// Mitsubishi GX Works2 project: Genova 14-11-2022_f1   PLC: FX1N/FX1NC

PROGRAM MAIN
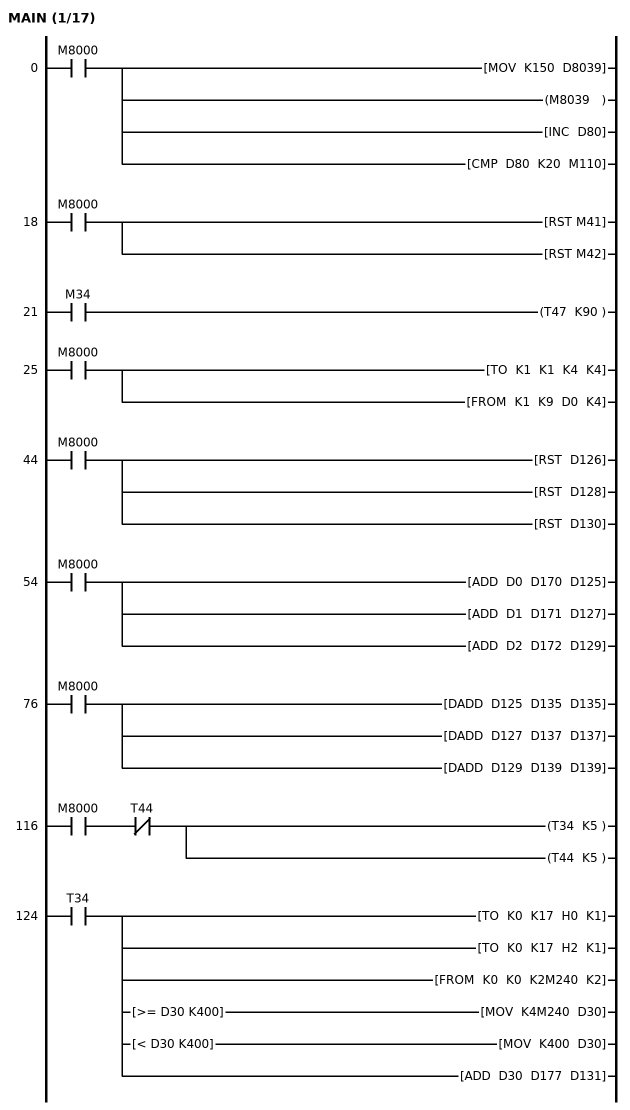
0     LD      M8000
      MOV     K150 D8039
      OUT     M8039
      INC     D80
      CMP     D80 K20 M110
18    LD      M8000
      RST     M41
      RST     M42
21    LD      M34
      OUT     T47 K90
25    LD      M8000
      TO      K1 K1 K4 K4
      FROM    K1 K9 D0 K4
44    LD      M8000
      RST     D126
      RST     D128
      RST     D130
54    LD      M8000
      ADD     D0 D170 D125
      ADD     D1 D171 D127
      ADD     D2 D172 D129
76    LD      M8000
      DADD    D125 D135 D135
      DADD    D127 D137 D137
      DADD    D129 D139 D139
116   LD      M8000
      ANI     T44
      OUT     T34 K5
      OUT     T44 K5
124   LD      T34
      TO      K0 K17 H0 K1
      TO      K0 K17 H2 K1
      FROM    K0 K0 K2M240 K2
      MPS
      AND>=   D30 K400
      MOV     K4M240 D30
      MRD
      AND<    D30 K400
      MOV     K400 D30
      MPP
      ADD     D30 D177 D131
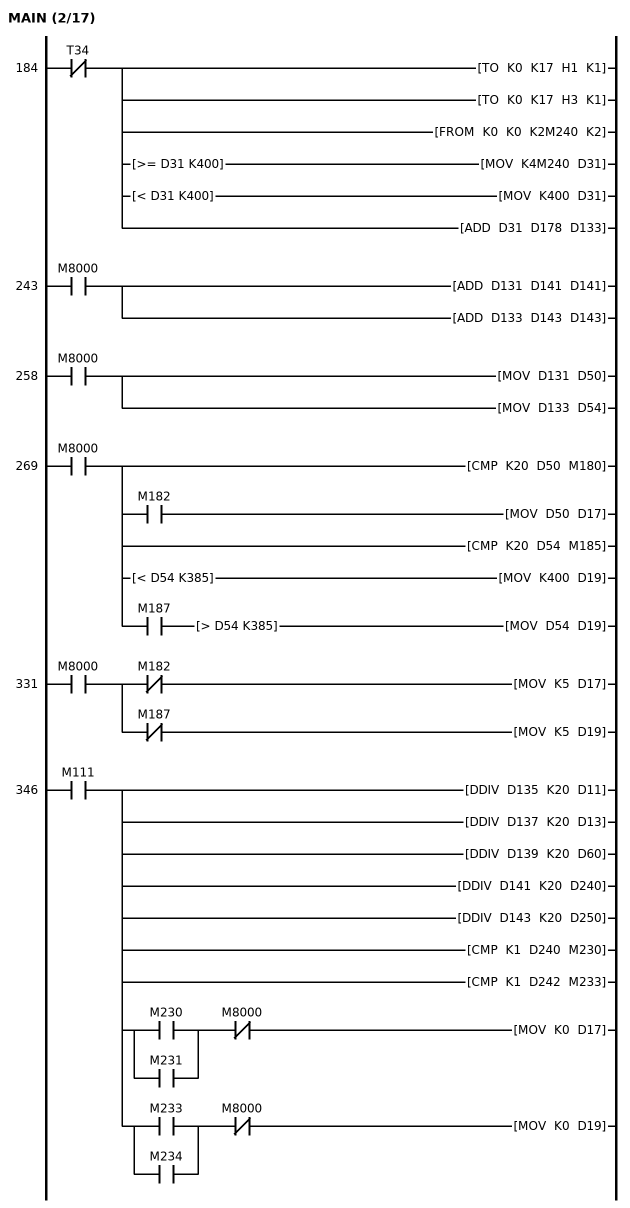
184   LDI     T34
      TO      K0 K17 H1 K1
      TO      K0 K17 H3 K1
      FROM    K0 K0 K2M240 K2
      MPS
      AND>=   D31 K400
      MOV     K4M240 D31
      MRD
      AND<    D31 K400
      MOV     K400 D31
      MPP
      ADD     D31 D178 D133
243   LD      M8000
      ADD     D131 D141 D141
      ADD     D133 D143 D143
258   LD      M8000
      MOV     D131 D50
      MOV     D133 D54
269   LD      M8000
      CMP     K20 D50 M180
      MPS
      AND     M182
      MOV     D50 D17
      MPP
      CMP     K20 D54 M185
      MPS
      AND<    D54 K385
      MOV     K400 D19
      MPP
      AND     M187
      AND>    D54 K385
      MOV     D54 D19
331   LD      M8000
      MPS
      ANI     M182
      MOV     K5 D17
      MPP
      ANI     M187
      MOV     K5 D19
346   LD      M111
      DDIV    D135 K20 D11
      DDIV    D137 K20 D13
      DDIV    D139 K20 D60
      DDIV    D141 K20 D240
      DDIV    D143 K20 D250
      CMP     K1 D240 M230
      CMP     K1 D242 M233
      MPS
      LD      M230
      OR      M231
      ANB
      ANI     M8000
      MOV     K0 D17
      MPP
      LD      M233
      OR      M234
      ANB
      ANI     M8000
      MOV     K0 D19
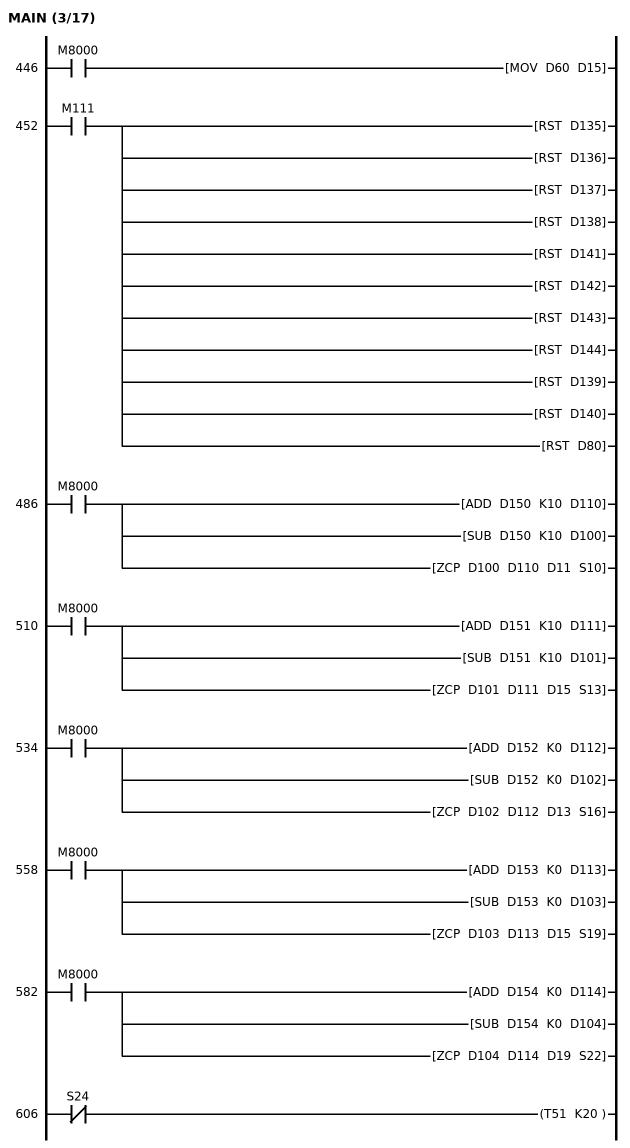
446   LD      M8000
      MOV     D60 D15
452   LD      M111
      RST     D135
      RST     D136
      RST     D137
      RST     D138
      RST     D141
      RST     D142
      RST     D143
      RST     D144
      RST     D139
      RST     D140
      RST     D80
486   LD      M8000
      ADD     D150 K10 D110
      SUB     D150 K10 D100
      ZCP     D100 D110 D11 S10
510   LD      M8000
      ADD     D151 K10 D111
      SUB     D151 K10 D101
      ZCP     D101 D111 D15 S13
534   LD      M8000
      ADD     D152 K0 D112
      SUB     D152 K0 D102
      ZCP     D102 D112 D13 S16
558   LD      M8000
      ADD     D153 K0 D113
      SUB     D153 K0 D103
      ZCP     D103 D113 D15 S19
582   LD      M8000
      ADD     D154 K0 D114
      SUB     D154 K0 D104
      ZCP     D104 D114 D19 S22
606   LDI     S24
      OUT     T51 K20
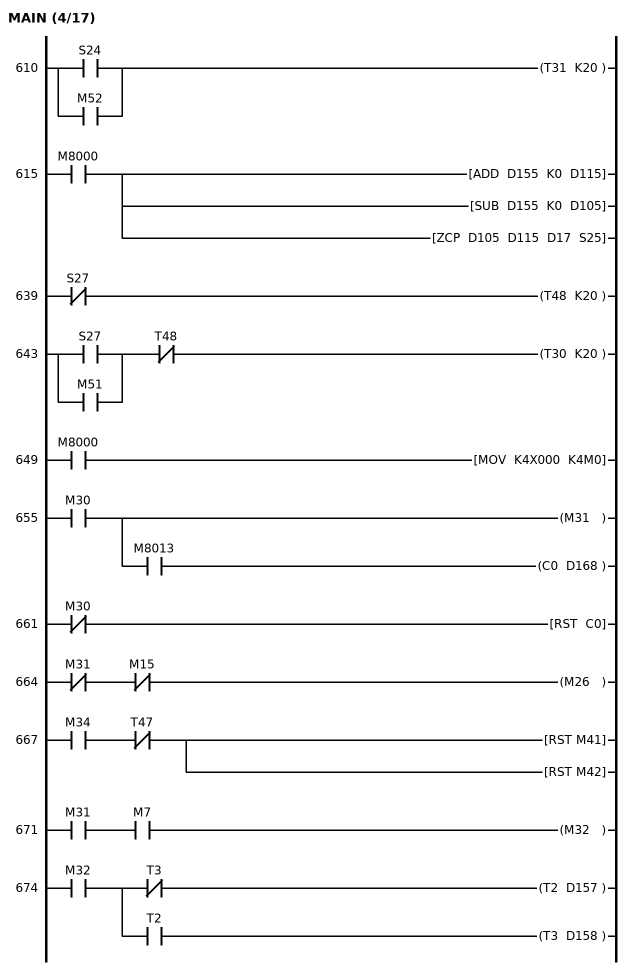
610   LD      S24
      OR      M52
      OUT     T31 K20
615   LD      M8000
      ADD     D155 K0 D115
      SUB     D155 K0 D105
      ZCP     D105 D115 D17 S25
639   LDI     S27
      OUT     T48 K20
643   LD      S27
      OR      M51
      ANI     T48
      OUT     T30 K20
649   LD      M8000
      MOV     K4X000 K4M0
655   LD      M30
      OUT     M31
      AND     M8013
      OUT     C0 D168
661   LDI     M30
      RST     C0
664   LDI     M31
      ANI     M15
      OUT     M26
667   LD      M34
      ANI     T47
      RST     M41
      RST     M42
671   LD      M31
      AND     M7
      OUT     M32
674   LD      M32
      MPS
      ANI     T3
      OUT     T2 D157
      MPP
      AND     T2
      OUT     T3 D158
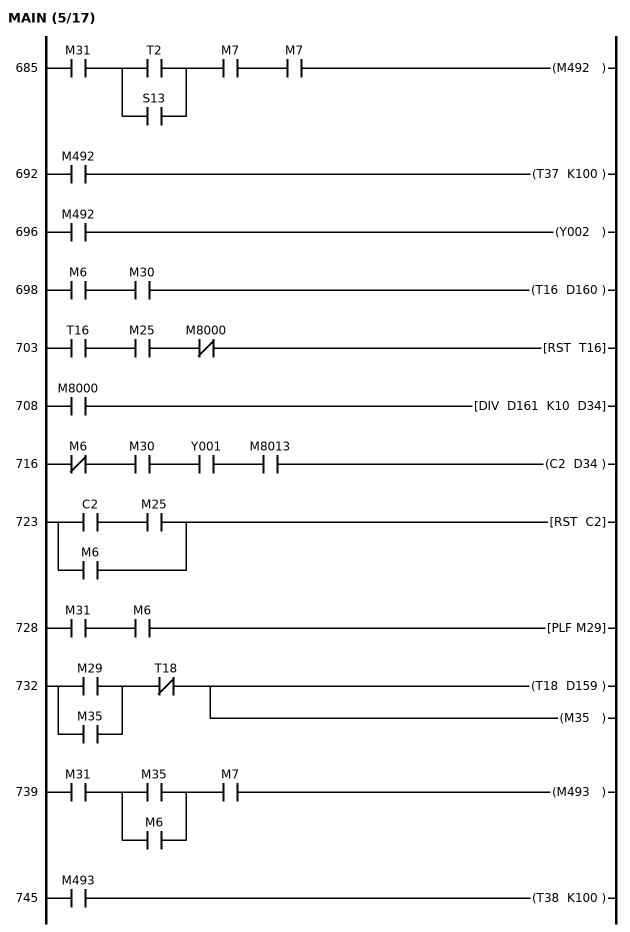
685   LD      M31
      LD      T2
      OR      S13
      ANB
      AND     M7
      AND     M7
      OUT     M492
692   LD      M492
      OUT     T37 K100
696   LD      M492
      OUT     Y002
698   LD      M6
      AND     M30
      OUT     T16 D160
703   LD      T16
      AND     M25
      ANI     M8000
      RST     T16
708   LD      M8000
      DIV     D161 K10 D34
716   LDI     M6
      AND     M30
      AND     Y001
      AND     M8013
      OUT     C2 D34
723   LD      C2
      AND     M25
      OR      M6
      RST     C2
728   LD      M31
      AND     M6
      PLF     M29
732   LD      M29
      OR      M35
      ANI     T18
      OUT     T18 D159
      OUT     M35
739   LD      M31
      LD      M35
      OR      M6
      ANB
      AND     M7
      OUT     M493
745   LD      M493
      OUT     T38 K100
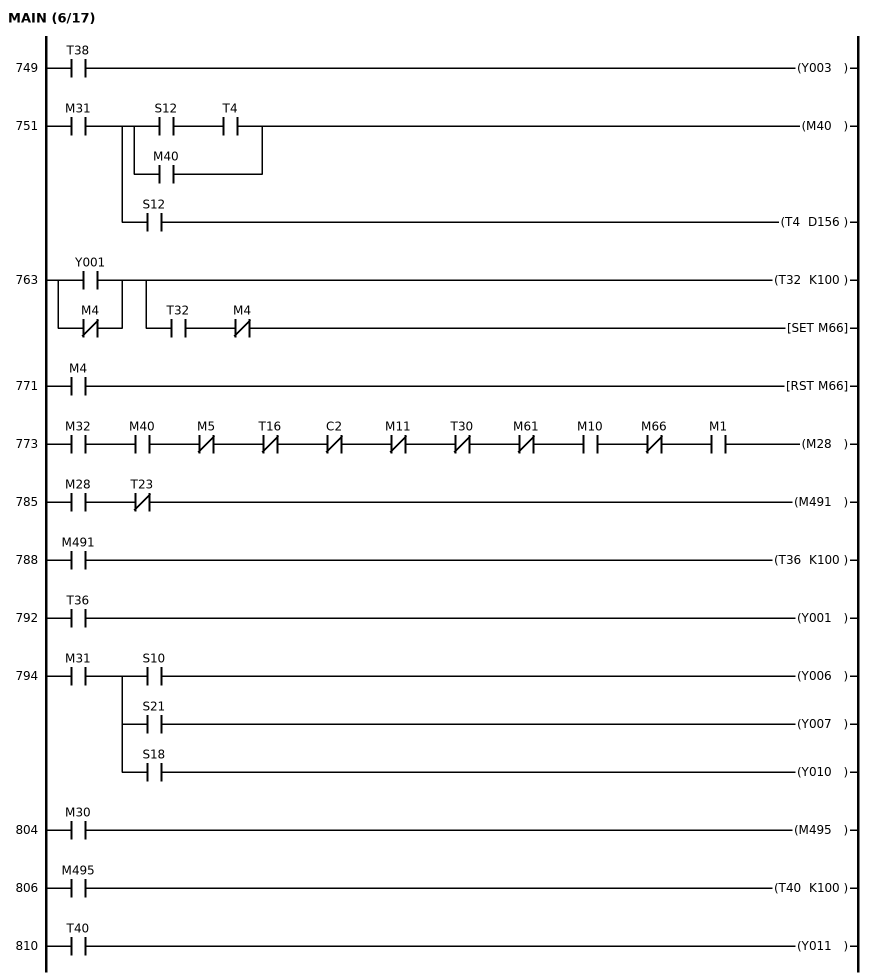
749   LD      T38
      OUT     Y003
751   LD      M31
      MPS
      LD      S12
      AND     T4
      OR      M40
      ANB
      OUT     M40
      MPP
      AND     S12
      OUT     T4 D156
763   LD      Y001
      ORI     M4
      OUT     T32 K100
      AND     T32
      ANI     M4
      SET     M66
771   LD      M4
      RST     M66
773   LD      M32
      AND     M40
      ANI     M5
      ANI     T16
      ANI     C2
      ANI     M11
      ANI     T30
      ANI     M61
      AND     M10
      ANI     M66
      AND     M1
      OUT     M28
785   LD      M28
      ANI     T23
      OUT     M491
788   LD      M491
      OUT     T36 K100
792   LD      T36
      OUT     Y001
794   LD      M31
      MPS
      AND     S10
      OUT     Y006
      MRD
      AND     S21
      OUT     Y007
      MPP
      AND     S18
      OUT     Y010
804   LD      M30
      OUT     M495
806   LD      M495
      OUT     T40 K100
810   LD      T40
      OUT     Y011
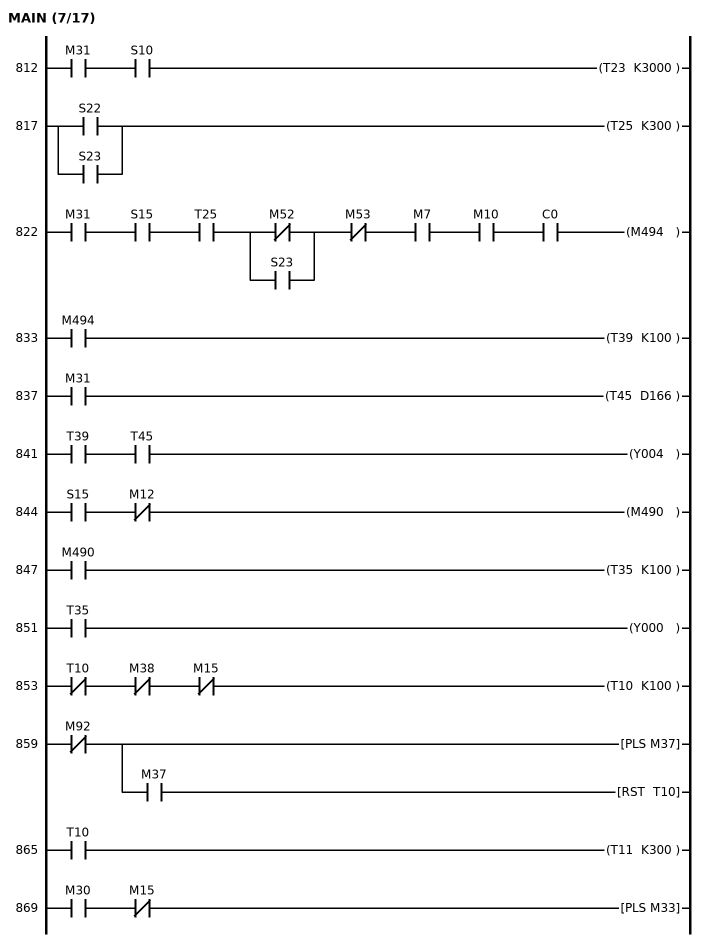
812   LD      M31
      AND     S10
      OUT     T23 K3000
817   LD      S22
      OR      S23
      OUT     T25 K300
822   LD      M31
      AND     S15
      AND     T25
      LDI     M52
      OR      S23
      ANB
      ANI     M53
      AND     M7
      AND     M10
      AND     C0
      OUT     M494
833   LD      M494
      OUT     T39 K100
837   LD      M31
      OUT     T45 D166
841   LD      T39
      AND     T45
      OUT     Y004
844   LD      S15
      ANI     M12
      OUT     M490
847   LD      M490
      OUT     T35 K100
851   LD      T35
      OUT     Y000
853   LDI     T10
      ANI     M38
      ANI     M15
      OUT     T10 K100
859   LDI     M92
      PLS     M37
      AND     M37
      RST     T10
865   LD      T10
      OUT     T11 K300
869   LD      M30
      ANI     M15
      PLS     M33
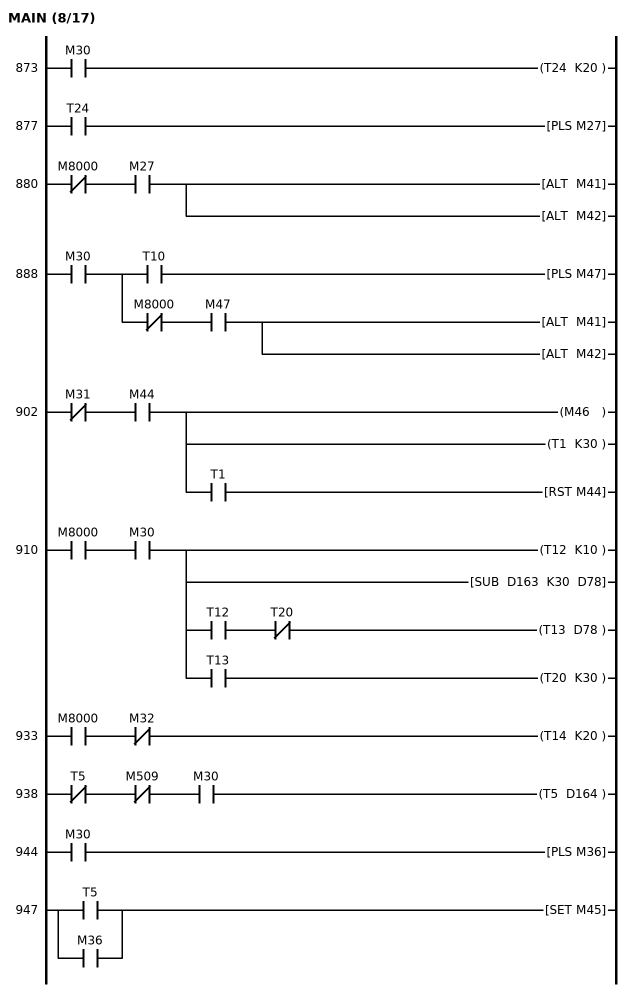
873   LD      M30
      OUT     T24 K20
877   LD      T24
      PLS     M27
880   LDI     M8000
      AND     M27
      ALT     M41
      ALT     M42
888   LD      M30
      MPS
      AND     T10
      PLS     M47
      MPP
      ANI     M8000
      AND     M47
      ALT     M41
      ALT     M42
902   LDI     M31
      AND     M44
      OUT     M46
      OUT     T1 K30
      AND     T1
      RST     M44
910   LD      M8000
      AND     M30
      OUT     T12 K10
      SUB     D163 K30 D78
      MPS
      AND     T12
      ANI     T20
      OUT     T13 D78
      MPP
      AND     T13
      OUT     T20 K30
933   LD      M8000
      ANI     M32
      OUT     T14 K20
938   LDI     T5
      ANI     M509
      AND     M30
      OUT     T5 D164
944   LD      M30
      PLS     M36
947   LD      T5
      OR      M36
      SET     M45
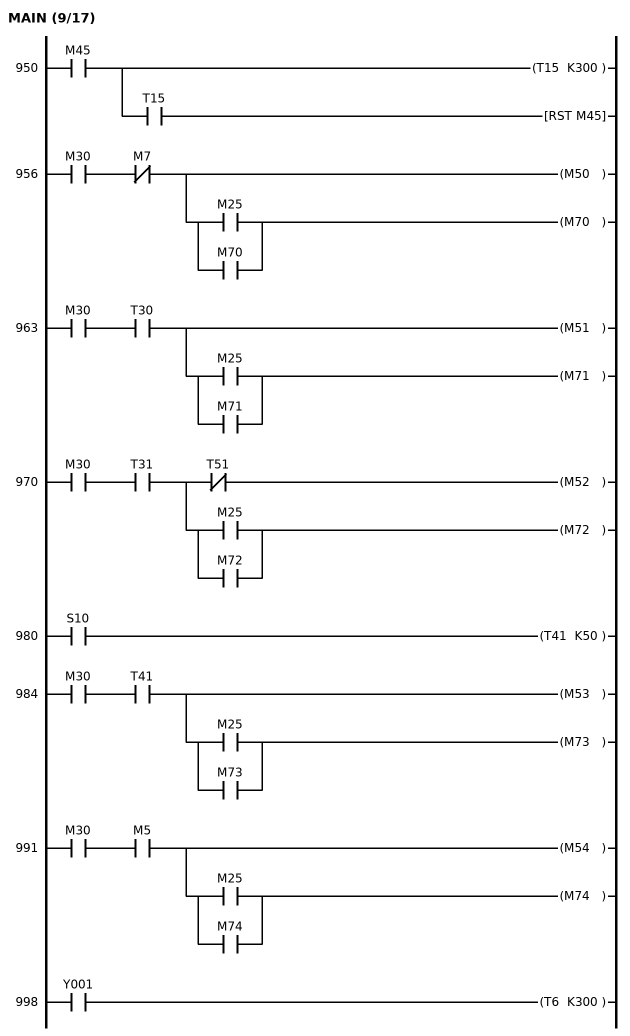
950   LD      M45
      OUT     T15 K300
      AND     T15
      RST     M45
956   LD      M30
      ANI     M7
      OUT     M50
      LD      M25
      OR      M70
      ANB
      OUT     M70
963   LD      M30
      AND     T30
      OUT     M51
      LD      M25
      OR      M71
      ANB
      OUT     M71
970   LD      M30
      AND     T31
      MPS
      ANI     T51
      OUT     M52
      MPP
      LD      M25
      OR      M72
      ANB
      OUT     M72
980   LD      S10
      OUT     T41 K50
984   LD      M30
      AND     T41
      OUT     M53
      LD      M25
      OR      M73
      ANB
      OUT     M73
991   LD      M30
      AND     M5
      OUT     M54
      LD      M25
      OR      M74
      ANB
      OUT     M74
998   LD      Y001
      OUT     T6 K300
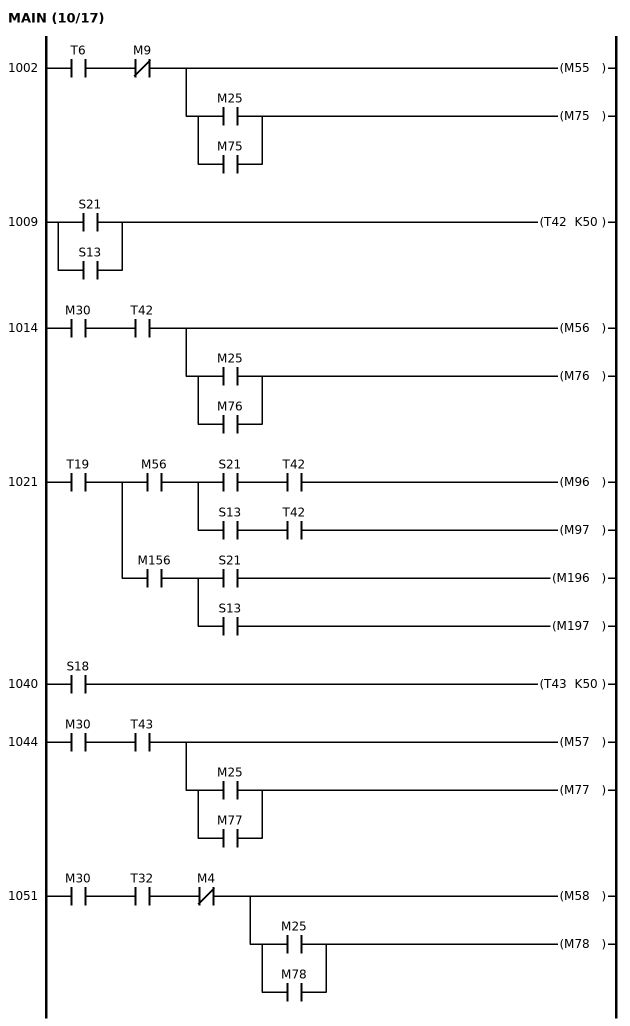
1002  LD      T6
      ANI     M9
      OUT     M55
      LD      M25
      OR      M75
      ANB
      OUT     M75
1009  LD      S21
      OR      S13
      OUT     T42 K50
1014  LD      M30
      AND     T42
      OUT     M56
      LD      M25
      OR      M76
      ANB
      OUT     M76
1021  LD      T19
      MPS
      AND     M56
      MPS
      AND     S21
      AND     T42
      OUT     M96
      MPP
      AND     S13
      AND     T42
      OUT     M97
      MPP
      AND     M156
      MPS
      AND     S21
      OUT     M196
      MPP
      AND     S13
      OUT     M197
1040  LD      S18
      OUT     T43 K50
1044  LD      M30
      AND     T43
      OUT     M57
      LD      M25
      OR      M77
      ANB
      OUT     M77
1051  LD      M30
      AND     T32
      ANI     M4
      OUT     M58
      LD      M25
      OR      M78
      ANB
      OUT     M78
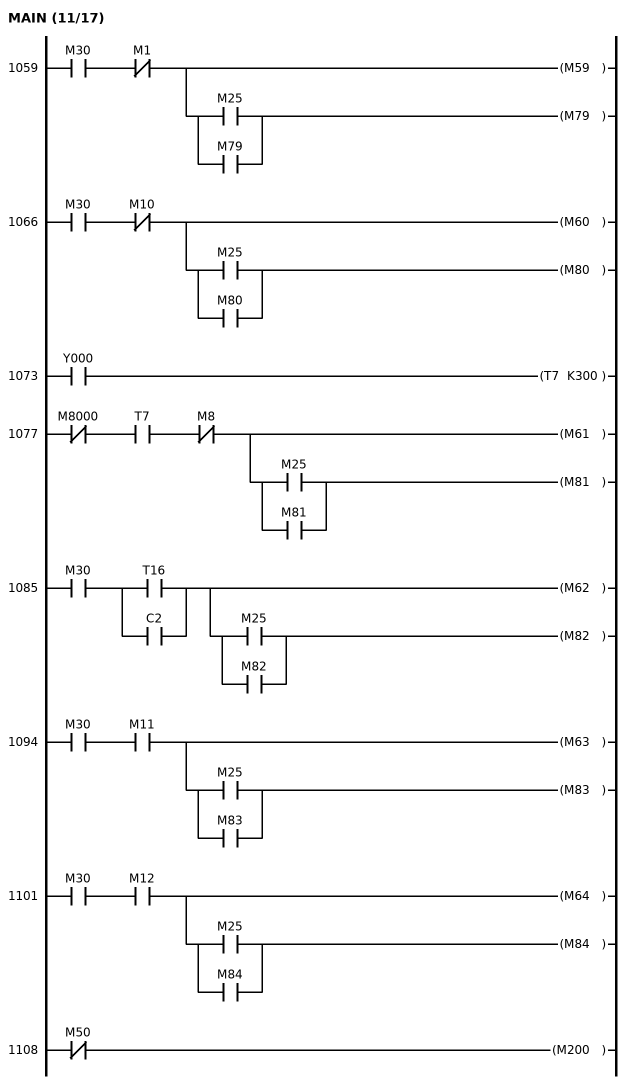
1059  LD      M30
      ANI     M1
      OUT     M59
      LD      M25
      OR      M79
      ANB
      OUT     M79
1066  LD      M30
      ANI     M10
      OUT     M60
      LD      M25
      OR      M80
      ANB
      OUT     M80
1073  LD      Y000
      OUT     T7 K300
1077  LDI     M8000
      AND     T7
      ANI     M8
      OUT     M61
      LD      M25
      OR      M81
      ANB
      OUT     M81
1085  LD      M30
      LD      T16
      OR      C2
      ANB
      OUT     M62
      LD      M25
      OR      M82
      ANB
      OUT     M82
1094  LD      M30
      AND     M11
      OUT     M63
      LD      M25
      OR      M83
      ANB
      OUT     M83
1101  LD      M30
      AND     M12
      OUT     M64
      LD      M25
      OR      M84
      ANB
      OUT     M84
1108  LDI     M50
      OUT     M200
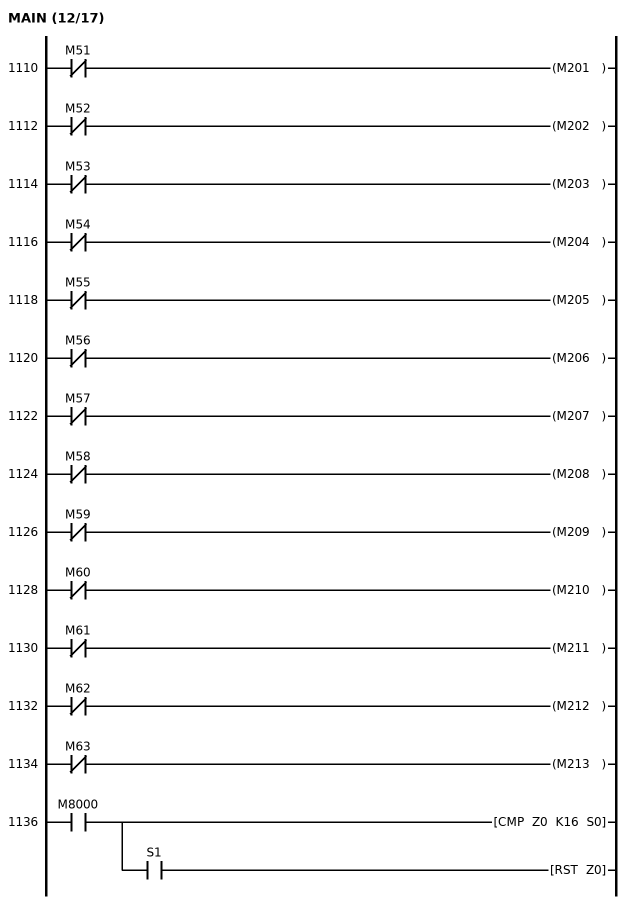
1110  LDI     M51
      OUT     M201
1112  LDI     M52
      OUT     M202
1114  LDI     M53
      OUT     M203
1116  LDI     M54
      OUT     M204
1118  LDI     M55
      OUT     M205
1120  LDI     M56
      OUT     M206
1122  LDI     M57
      OUT     M207
1124  LDI     M58
      OUT     M208
1126  LDI     M59
      OUT     M209
1128  LDI     M60
      OUT     M210
1130  LDI     M61
      OUT     M211
1132  LDI     M62
      OUT     M212
1134  LDI     M63
      OUT     M213
1136  LD      M8000
      CMP     Z0 K16 S0
      AND     S1
      RST     Z0
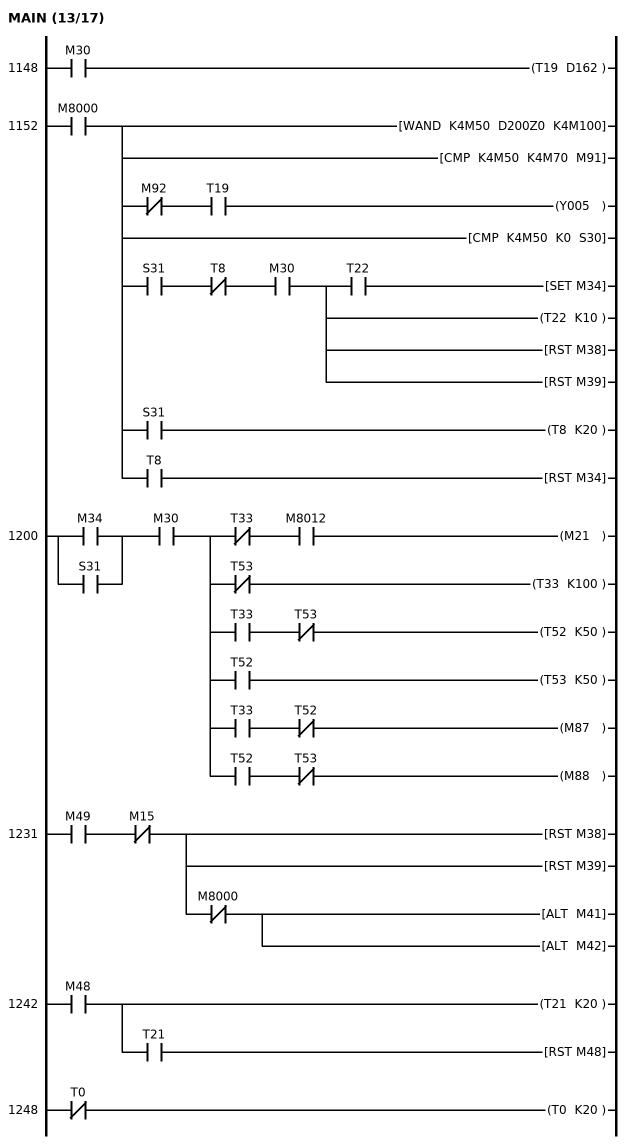
1148  LD      M30
      OUT     T19 D162
1152  LD      M8000
      WAND    K4M50 D200Z0 K4M100
      CMP     K4M50 K4M70 M91
      MPS
      ANI     M92
      AND     T19
      OUT     Y005
      MPP
      CMP     K4M50 K0 S30
      MPS
      AND     S31
      ANI     T8
      AND     M30
      MPS
      AND     T22
      SET     M34
      MPP
      OUT     T22 K10
      RST     M38
      RST     M39
      MRD
      AND     S31
      OUT     T8 K20
      MPP
      AND     T8
      RST     M34
1200  LD      M34
      OR      S31
      AND     M30
      MPS
      ANI     T33
      AND     M8012
      OUT     M21
      MRD
      ANI     T53
      OUT     T33 K100
      MRD
      AND     T33
      ANI     T53
      OUT     T52 K50
      MRD
      AND     T52
      OUT     T53 K50
      MRD
      AND     T33
      ANI     T52
      OUT     M87
      MPP
      AND     T52
      ANI     T53
      OUT     M88
1231  LD      M49
      ANI     M15
      RST     M38
      RST     M39
      ANI     M8000
      ALT     M41
      ALT     M42
1242  LD      M48
      OUT     T21 K20
      AND     T21
      RST     M48
1248  LDI     T0
      OUT     T0 K20
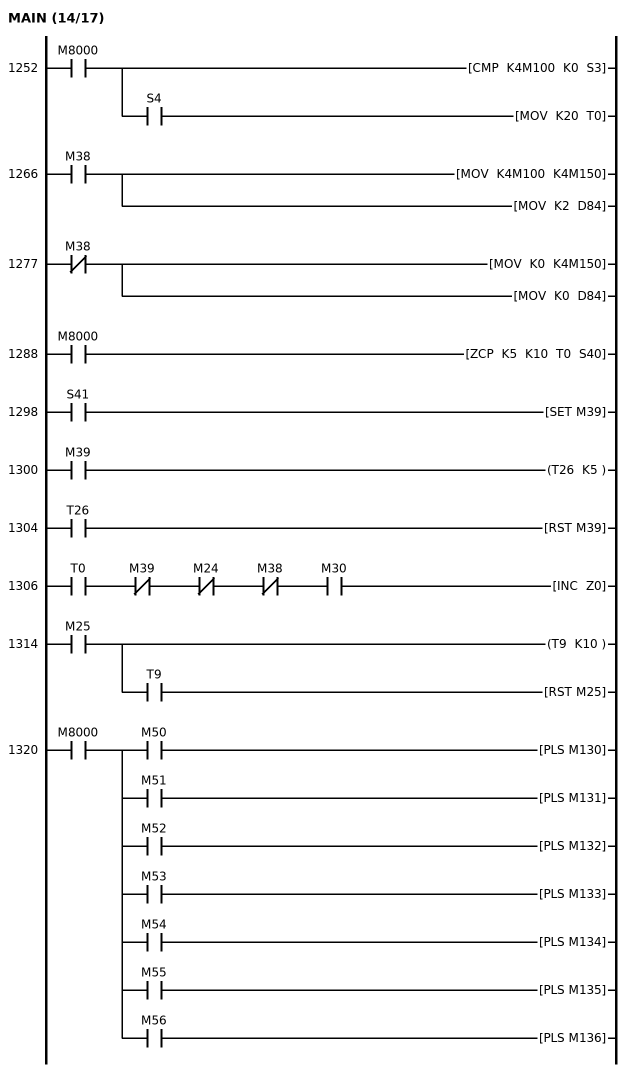
1252  LD      M8000
      CMP     K4M100 K0 S3
      AND     S4
      MOV     K20 T0
1266  LD      M38
      MOV     K4M100 K4M150
      MOV     K2 D84
1277  LDI     M38
      MOV     K0 K4M150
      MOV     K0 D84
1288  LD      M8000
      ZCP     K5 K10 T0 S40
1298  LD      S41
      SET     M39
1300  LD      M39
      OUT     T26 K5
1304  LD      T26
      RST     M39
1306  LD      T0
      ANI     M39
      ANI     M24
      ANI     M38
      AND     M30
      INC     Z0
1314  LD      M25
      OUT     T9 K10
      AND     T9
      RST     M25
1320  LD      M8000
      MPS
      AND     M50
      PLS     M130
      MRD
      AND     M51
      PLS     M131
      MRD
      AND     M52
      PLS     M132
      MRD
      AND     M53
      PLS     M133
      MRD
      AND     M54
      PLS     M134
      MRD
      AND     M55
      PLS     M135
      MPP
      AND     M56
      PLS     M136
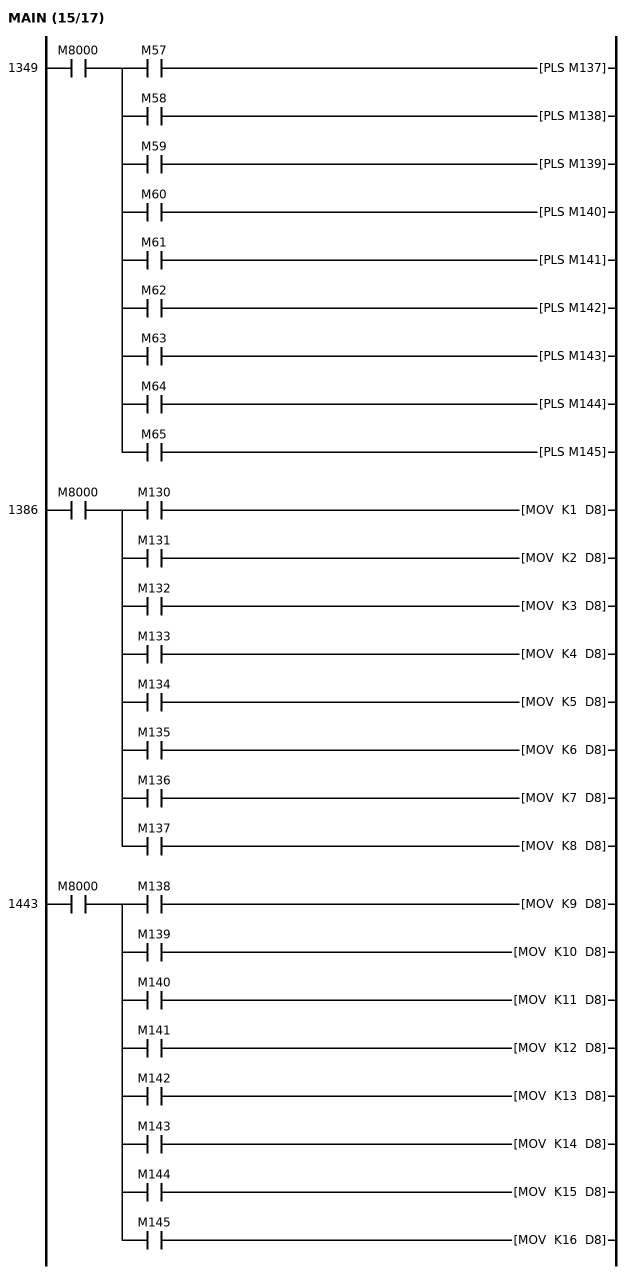
1349  LD      M8000
      MPS
      AND     M57
      PLS     M137
      MRD
      AND     M58
      PLS     M138
      MRD
      AND     M59
      PLS     M139
      MRD
      AND     M60
      PLS     M140
      MRD
      AND     M61
      PLS     M141
      MRD
      AND     M62
      PLS     M142
      MRD
      AND     M63
      PLS     M143
      MRD
      AND     M64
      PLS     M144
      MPP
      AND     M65
      PLS     M145
1386  LD      M8000
      MPS
      AND     M130
      MOV     K1 D8
      MRD
      AND     M131
      MOV     K2 D8
      MRD
      AND     M132
      MOV     K3 D8
      MRD
      AND     M133
      MOV     K4 D8
      MRD
      AND     M134
      MOV     K5 D8
      MRD
      AND     M135
      MOV     K6 D8
      MRD
      AND     M136
      MOV     K7 D8
      MPP
      AND     M137
      MOV     K8 D8
1443  LD      M8000
      MPS
      AND     M138
      MOV     K9 D8
      MRD
      AND     M139
      MOV     K10 D8
      MRD
      AND     M140
      MOV     K11 D8
      MRD
      AND     M141
      MOV     K12 D8
      MRD
      AND     M142
      MOV     K13 D8
      MRD
      AND     M143
      MOV     K14 D8
      MRD
      AND     M144
      MOV     K15 D8
      MPP
      AND     M145
      MOV     K16 D8
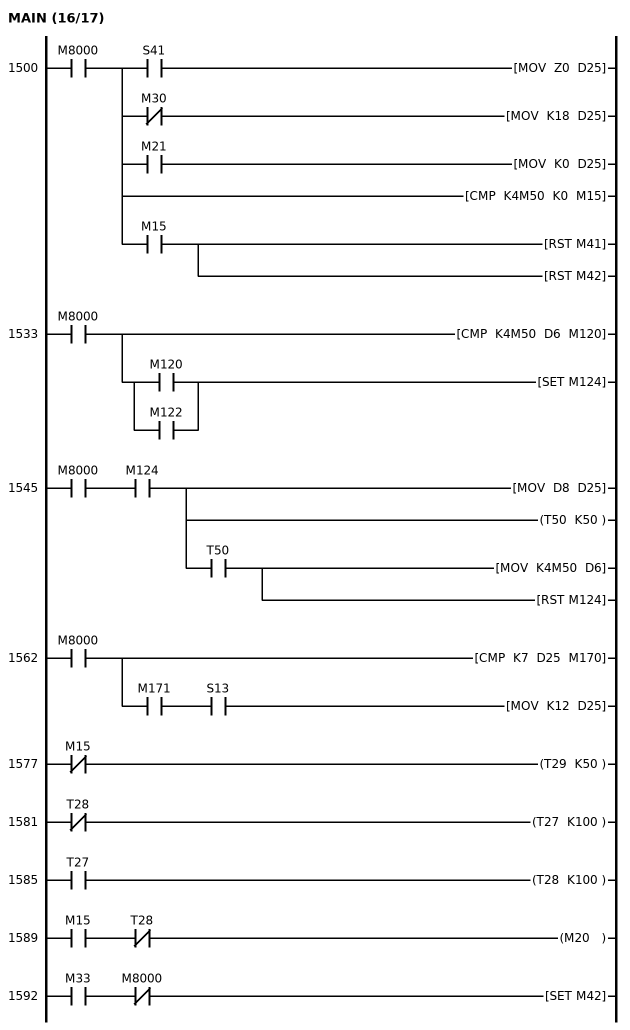
1500  LD      M8000
      MPS
      AND     S41
      MOV     Z0 D25
      MRD
      ANI     M30
      MOV     K18 D25
      MRD
      AND     M21
      MOV     K0 D25
      MPP
      CMP     K4M50 K0 M15
      AND     M15
      RST     M41
      RST     M42
1533  LD      M8000
      CMP     K4M50 D6 M120
      LD      M120
      OR      M122
      ANB
      SET     M124
1545  LD      M8000
      AND     M124
      MOV     D8 D25
      OUT     T50 K50
      AND     T50
      MOV     K4M50 D6
      RST     M124
1562  LD      M8000
      CMP     K7 D25 M170
      AND     M171
      AND     S13
      MOV     K12 D25
1577  LDI     M15
      OUT     T29 K50
1581  LDI     T28
      OUT     T27 K100
1585  LD      T27
      OUT     T28 K100
1589  LD      M15
      ANI     T28
      OUT     M20
1592  LD      M33
      ANI     M8000
      SET     M42
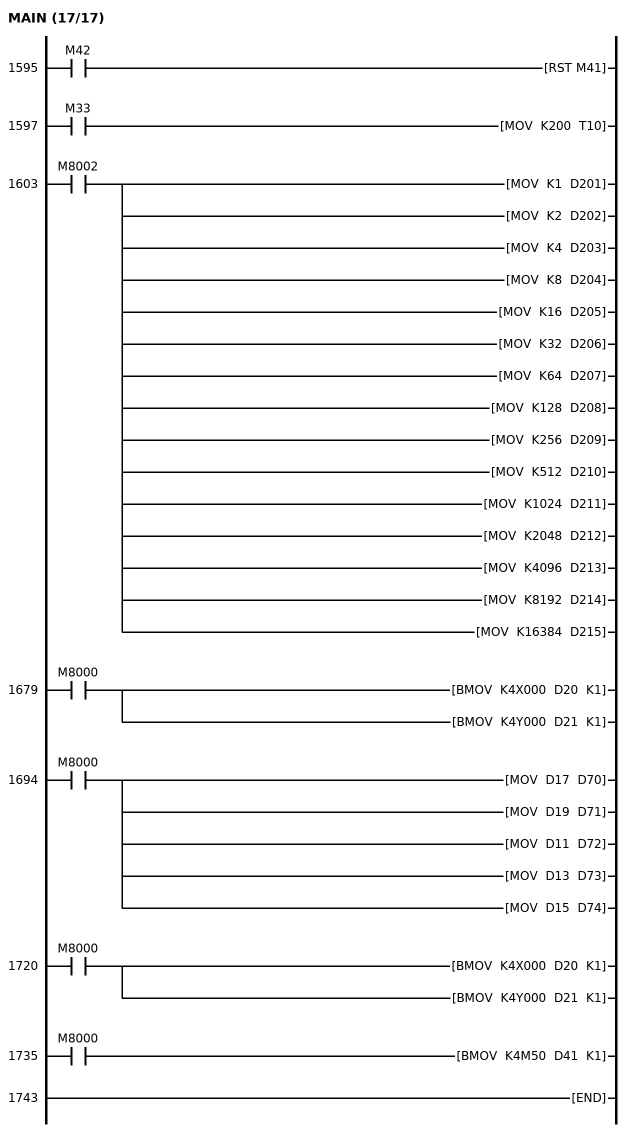
1595  LD      M42
      RST     M41
1597  LD      M33
      MOV     K200 T10
1603  LD      M8002
      MOV     K1 D201
      MOV     K2 D202
      MOV     K4 D203
      MOV     K8 D204
      MOV     K16 D205
      MOV     K32 D206
      MOV     K64 D207
      MOV     K128 D208
      MOV     K256 D209
      MOV     K512 D210
      MOV     K1024 D211
      MOV     K2048 D212
      MOV     K4096 D213
      MOV     K8192 D214
      MOV     K16384 D215
1679  LD      M8000
      BMOV    K4X000 D20 K1
      BMOV    K4Y000 D21 K1
1694  LD      M8000
      MOV     D17 D70
      MOV     D19 D71
      MOV     D11 D72
      MOV     D13 D73
      MOV     D15 D74
1720  LD      M8000
      BMOV    K4X000 D20 K1
      BMOV    K4Y000 D21 K1
1735  LD      M8000
      BMOV    K4M50 D41 K1
1743  END
END_PROGRAM
